(* IEC 61131-3 sources: learning-path/04_introduction_to_st/exercises/4_timer_for_tank/src, 2 files *)

(* ---- valve.st ---- *)
NAMESPACE Siemens.AxTraining.ControlModules

    FUNCTION_BLOCK Valve
        VAR_INPUT
            cmdOpen :BOOL;
            cmdClose: BOOL;
        END_VAR
        VAR_OUTPUT
            ctrlOpen :BOOL;
            ctrlClose : BOOL;
        END_VAR

        ctrlClose := FALSE;
        ctrlOpen := FALSE;

        IF cmdClose THEN
            ctrlClose := TRUE;
        ELSIF cmdOpen THEN
            ctrlOpen := TRUE;
        END_IF;

    END_FUNCTION_BLOCK

END_NAMESPACE

(* ---- configuration.st ---- *)
USING Siemens.AxTraining;
CONFIGURATION PLC_1
    TASK Main(Interval := T#10ms, Priority := 1);
    PROGRAM P1 WITH Main: FluidProgram;

    VAR_GLOBAL
        enableTank : BOOL;
        inletOpenTank : BOOL;
        outletOpenTank : BOOL;
    END_VAR
END_CONFIGURATION
